PROGRAM MAIN
VAR
	blueEdgeDetector : EdgeDetectorWithDoubleTap;
	
END_VAR

END_PROGRAM

(* stored: Version 1.1.0.1, ProductVersion 3.1.4022.10
   POU MAIN: Id {22a0f490-9a43-4d76-8f19-31a50310cd0f}, SpecialFunc None *)
